{attribute 'GeneratedUsingTerminal: EL7332-0000-0016'}
{attribute addProperty BoxType "EL7332-0000-0016"}
{attribute addProperty Id "StatusAT %I*Status_B679584511"}
{attribute addProperty CRC "921504111"}
{attribute addProperty Size "11"}
TYPE DCM_Status_Channel_36ED096F :
STRUCT
	{attribute addProperty Name "Status"}
	Status AT %I* : Status_B6795845;
END_STRUCT
END_TYPE

(* stored: Version 1.2.0.0, ProductVersion 3.1.4024.9
   DUT DCM_Status_Channel_36ED096F: Id {2b2886c8-2298-41c9-bc44-fcc071e03667} *)
